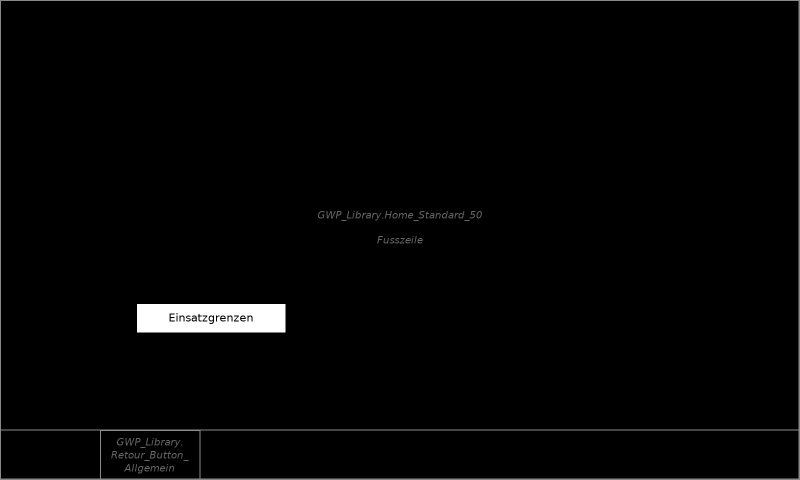
VISUALIZATION Home  // 800x480
    Frame (0,0 800x430)
        shows GWP_Library.Home_Standard_50()
    Rectangle (136,303 150x30), "Einsatzgrenzen"
        OnMouseClick: change screen: EG
    Frame (0,0 800x480)
        shows Fusszeile()
    Frame (100,430 100x50)
        shows GWP_Library.Retour_Button_Allgemein()
END_VISUALIZATION

(* stored: Version 1.1.0.1, ProductVersion 3.1.4022.6
   Visu Home: Id {033fb334-df85-464e-8ac8-1b8037b57141} *)
